// TIA Portal V17 export
// export: Created 2024-08-20T10:59:42.3933613Z, ExportSetting WithDefaults, DisplayName Totally Integrated Automation Portal, DisplayVersion V17 Update 4, DisplayName TIA Portal Openness, DisplayVersion V17 Update 4, DisplayName TIA Portal Version Control Interface, DisplayVersion V17, DisplayName STEP 7 Professional, DisplayVersion V17 Update 4, DisplayName STEP 7 Safety, DisplayVersion V17, DisplayName WinCC Advanced, DisplayVersion V17 Update 4
DATA_BLOCK "DIVERSOS"   // DB1
{ S7_Optimized_Access := 'TRUE' }
VERSION : 0.1
// stored: AutoNumber false, DBAccessibleFromOPCUA true, IsOnlyStoredInLoadMemory false, IsRetainMemResEnabled false, IsWriteProtectedInAS false, MemoryReserve 100
   VAR
      T1S : Bool;   // PULSO A CADA 1 SEGUNDO
      AUX_T1S : Bool;   // PULSO A CADA 1 SEGUNDO
      QTDE_PULSO : DInt := 200;
      ForcePulso : Bool;
      N_L00P : Int;
      Aux_N_LOOP : Int;
      Looping : Int := 0;
      TMR : Array[0..10] of IEC_TIMER;
      P1S { S7_SetPoint := 'True'} : Bool;   // Pulso de 1 segundo
      "MB-01-SP" : Bool;   // Solicitação partida de bomba
      "MB-02-SP" : Bool;   // Solicitação partida de bomba
      "MB-03-SP" : Bool;   // Solicitação partida de bomba
      "MB-04-SP" : Bool;   // Solicitação partida de bomba
   END_VAR
BEGIN
END_DATA_BLOCK
